PROGRAM MAIN
VAR_OUTPUT
	currentTime : TIMESTRUCT;
END_VAR
VAR
	sMessage : STRING := 'from SERVER to CLIENT';
	newRecipient : STRING;
	newData : AdsData;
	retrievedData : AdsData;
	
	sendOnce : BOOL;
	sendFastNum : BOOL;
	
	i : INT := 0;
	
	fbLocalSystemTime : FB_LocalSystemTime;
END_VAR

IF NOT setup() THEN
	RETURN;
END_IF

AdsTcp_WinStd(
	bBusy=> , 
	err=> , 
	errid=> , 
	areaSockets=> );
	
IF sendOnce OR sendFastNum THEN
	MEMSET(ADR(newData), 0, SIZEOF(newData));
	
	sMessage := TO_STRING(i);
	
	newRecipient := TO_STRING(AreaNum.AREA_2);
	newData.description := EventsEnum.TEST_COMMS;
	newData.timestamp := currentTime;
	MEMCPY(ADR(newData.binaryData), ADR(sMessage), LEN(sMessage));
	
	AdsTcp_WinStd.queueMessage(recipient := newRecipient, data := newData);
	
	i := i + 1;
	sendOnce := FALSE;
END_IF

retrievedData := AdsTcp_WinStd.AREA_2.receivingData;

METHOD setup : BOOL
VAR
END_VAR
fbLocalSystemTime(
	sNetID:= , 
	bEnable:= TRUE, 
	dwCycle:= , 
	dwOpt:= , 
	tTimeout:= , 
	bValid=> , 
	systemTime=> currentTime, 
	tzID=> );

setup := TRUE;
END_METHOD

END_PROGRAM

(* stored: Version 1.1.0.1, ProductVersion 3.1.4024.11
   POU MAIN: Id {2cbdba0c-ad31-4c75-8f6b-289818655c29}, SpecialFunc None
   Method setup: Id {60067628-0974-47f6-84ab-860dda211b04} *)
